INTERFACE I_FileAccess

PROPERTY FileProperties : REFERENCE TO ST_FileProperties
GET
END_GET
SET
END_SET
END_PROPERTY

END_INTERFACE

(* stored: Version 1.1.0.1, ProductVersion 3.1.4024.13
   Itf I_FileAccess: Id {f6e2d3cb-8903-0f1f-08af-c71e2f897578}
   Property FileProperties: Id {3d266cd2-f99a-09d0-2792-cabadc23f86c}
   Get Get: Id {bc2f37ba-44fe-0293-08d8-3751aba78ca4}
   Set Set: Id {1598fe0c-3ad1-069f-0d89-cc518d0d2342} *)
